TYPE XTSCommands_typ :
    STRUCT

        Enable  : BOOL; // Enables Movers & Collision Avoidance, activates M1 Detection

    END_STRUCT
END_TYPE

(* stored: Version 1.1.0.1, ProductVersion 3.1.4026.8
   DUT XTSCommands_typ: Id {dc2a4f5e-f09b-4e87-82b1-79343e5d1394} *)
